Fanuc KAREL source: kf00075.KL

-- PROVISIONAL review KL for V940-1; original PC SHA256 9d042b4ccbc4f79fee4dc0f77e958b936716819a140df87833a0242e5d76ee3a
-- Incomplete behavior may be omitted. Consult companion uncertainty JSON. Do not deploy.
PROGRAM KF00075
%NOLOCKGROUP
VAR
  I : INTEGER
  J : INTEGER
  X : REAL
  Y : REAL
  B : BOOLEAN
  C : BOOLEAN
  TXT : STRING[80]
  TXT2 : STRING[80]
  STATUS : INTEGER
-- UNRESOLVED_DECL AI type=002010
-- UNRESOLVED_DECL BI type=002010
-- UNRESOLVED_DECL P type=000102
-- UNRESOLVED_DECL JP type=000199
-- UNRESOLVED_DECL PF type=000101
-- UNRESOLVED_DECL V1 type=000013
-- UNRESOLVED_DECL V2 type=000013
BEGIN
  -- V9_ZERO_TABLE_METADATA_HINT layout=0001; no indexed target words; source/name/runtime held
  -- UNRESOLVED_PC offsets 5-15; opcodes 3F,75
  -- UNRESOLVED_PC offsets 20-29; opcodes 3F,75
  -- UNRESOLVED_PC offsets 34-45; opcodes 2E,23
  -- UNRESOLVED_PC offsets 50-61; opcodes 2E,23
  -- UNRESOLVED_PC offsets 66-85; opcodes 27,22,2A,27,9D,76,23
  -- UNRESOLVED_PC offsets 90-94; opcodes 7F
END KF00075
